// TIA Portal V17 export
// export: Created 2023-12-22T15:03:09.492741Z, ExportSetting WithDefaults, DisplayName Totally Integrated Automation Portal, DisplayVersion V17, DisplayName TIA Portal Openness, DisplayVersion V17, DisplayName TIA Portal Version Control Interface, DisplayVersion V17, DisplayName STEP 7 Professional, DisplayVersion V17, DisplayName STEP 7 Safety, DisplayVersion V17, DisplayName WinCC Advanced, DisplayVersion V17
DATA_BLOCK "tGw_DB"   // DB3
{ S7_Optimized_Access := 'TRUE' }
VERSION : 0.1
// stored: AutoNumber true, DBAccessibleFromOPCUA true, DBAccessibleFromWebserver true, IsOnlyStoredInLoadMemory false, IsRetainMemResEnabled false, IsWriteProtectedInAS false, MemoryReserve 100
   VAR RETAIN
      tGw : Array[0..31] of Struct   // Точка подключения к КП
         IP { S7_SetPoint := 'True'} : IP_V4;
         Port { S7_SetPoint := 'True'} : UInt;
      END_STRUCT;
   END_VAR
BEGIN
   tGw[0].IP.ADDR[1] := 16#0A;
   tGw[0].IP.ADDR[2..3] := 16#01;
   tGw[0].IP.ADDR[4] := 16#9B;
   tGw[1].IP.ADDR[1] := 16#0A;
   tGw[1].IP.ADDR[2..3] := 16#01;
   tGw[1].IP.ADDR[4] := 16#C9;
   tGw[2].IP.ADDR[1] := 16#0A;
   tGw[2].IP.ADDR[2..3] := 16#01;
   tGw[2].IP.ADDR[4] := 16#CA;
   tGw[3].IP.ADDR[1] := 16#0A;
   tGw[3].IP.ADDR[2..3] := 16#01;
   tGw[3].IP.ADDR[4] := 16#CB;
   tGw[4].IP.ADDR[1] := 16#0A;
   tGw[4].IP.ADDR[2..3] := 16#01;
   tGw[4].IP.ADDR[4] := 16#D4;
   tGw[5].IP.ADDR[1] := 16#0A;
   tGw[5].IP.ADDR[2..3] := 16#01;
   tGw[5].IP.ADDR[4] := 16#D5;
   tGw[6].IP.ADDR[1] := 16#0A;
   tGw[6].IP.ADDR[2..3] := 16#01;
   tGw[6].IP.ADDR[4] := 16#D6;
   tGw[7].IP.ADDR[1] := 16#0A;
   tGw[7].IP.ADDR[2..3] := 16#01;
   tGw[7].IP.ADDR[4] := 16#D7;
   tGw[8].IP.ADDR[1] := 16#0A;
   tGw[8].IP.ADDR[2..3] := 16#01;
   tGw[8].IP.ADDR[4] := 16#DC;
   tGw[9].IP.ADDR[1] := 16#0A;
   tGw[9].IP.ADDR[2..3] := 16#01;
   tGw[9].IP.ADDR[4] := 16#DD;
   tGw[10].IP.ADDR[1] := 16#0A;
   tGw[10].IP.ADDR[2..3] := 16#01;
   tGw[10].IP.ADDR[4] := 16#DE;
   tGw[11].IP.ADDR[1] := 16#0A;
   tGw[11].IP.ADDR[2..3] := 16#01;
   tGw[11].IP.ADDR[4] := 16#DF;
   tGw[0..11].Port := 504;
   tGw[12].Port := 502;
   tGw[13].Port := 503;
   tGw[14].Port := 504;
   tGw[15].Port := 502;
   tGw[16].Port := 503;
   tGw[17].Port := 504;
   tGw[18..21].Port := 502;
   tGw[22..31].Port := 0;
END_DATA_BLOCK
